FUNCTION_BLOCK FB_CommandInvoker
VAR_GENERIC CONSTANT
	CommandCapacity : UINT := 10;
END_VAR
EXTENDS FB_Base
VAR
	_Commands : ARRAY[0..CommandCapacity - 1] OF I_Command;
	_CommandCount : UINT;
	
	_InvokeIndex : UINT;
	_ProgressState : E_Progress;
	
	_PauseRequest : BOOL;
	_StepMode : BOOL;
END_VAR

METHOD AddCommand : BOOL
VAR_INPUT
	command : I_Command;
END_VAR
IF (NOT _CommandCount < CommandCapacity) THEN
	Tc2_System.ADSLOGSTR(0, 'Can not add any more commands!', '');
	RETURN;
END_IF

_Commands[_CommandCount] := command;
_CommandCount := _CommandCount + 1;

AddCommand := TRUE;
END_METHOD

METHOD ClearCommands
VAR
	i : UINT;
	p : POINTER TO BYTE;
END_VAR
FOR i := 0 TO _CommandCount - 1 DO
	__QUERYPOINTER(_Commands[i], p);
	__DELETE(p);
END_FOR

_CommandCount := 0;
END_METHOD

{attribute 'monitoring' := 'call'}
PROPERTY CommandCount : UINT
GET
CommandCount := _CommandCount;
END_GET
END_PROPERTY

{attribute 'monitoring' := 'call'}
PROPERTY Commands : REFERENCE TO ARRAY[0..CommandCapacity - 1] OF I_Command
GET
Commands REF= _Commands;
END_GET
END_PROPERTY

METHOD Cyclic
VAR_INPUT
END_VAR
IF (_ProgressState = E_Progress.Running) THEN
	Invoke();
END_IF
END_METHOD

//FB_Exit must be implemented explicitly. If there is an implementation, then the
//method is called before the controller removes the code of the function block instance
//(implicit call). The return value is not evaluated.
METHOD FB_Exit: BOOL
VAR_INPUT
    bInCopyCode: BOOL;  // TRUE: the exit method is called in order to leave the instance which will be copied afterwards (online change).  
END_VAR
ClearCommands();
END_METHOD

METHOD PRIVATE Invoke
VAR
	commandProgress : E_Progress;
	progress : T_MaxString;
	test : STRING := 'test';
END_VAR
IF (_CommandCount = 0) THEN
	_ProgressState := E_Progress.Completed;
	
	Tc2_System.ADSLOGSTR(0, 'Invoker finished. No commands were executed.', '');	
END_IF

IF (_InvokeIndex < _CommandCount) THEN
	
	commandProgress := _Commands[_InvokeIndex].Execute();
	IF (commandProgress = E_Progress.Completed) THEN
		
		IF (_PauseRequest OR _StepMode) THEN
			_ProgressState := E_Progress.Paused;
			_PauseRequest := FALSE;
		END_IF
		
		IF (_InvokeIndex = _CommandCount - 1) THEN
			_ProgressState := E_Progress.Completed;
			
			Tc2_System.ADSLOGSTR(0, 'Invoker finished', '');
		END_IF

		_InvokeIndex := _InvokeIndex + 1;
		
		progress := 'Invoker progress  ';
		progress := CONCAT(progress, TO_STRING(_InvokeIndex));
		progress := CONCAT(progress, '/');
		progress := CONCAT(progress, TO_STRING(_CommandCount));
		progress := CONCAT(progress, '  ');
		progress := CONCAT(progress, LREAL_TO_FMTSTR(ProgressPercent, 1, TRUE));
		progress := CONCAT(progress, ' %s');
		Tc2_System.ADSLOGSTR(0, progress, '%');
// 		Tc2_System.ADSLOGSTR(0, 'ahoj', '');
// 		Tc2_System.ADSLOGSTR(0, progress, '');
	END_IF
END_IF
END_METHOD

{attribute 'monitoring' := 'call'}
PROPERTY InvokeIndex : UINT
GET
InvokeIndex := _InvokeIndex;
END_GET
END_PROPERTY

METHOD Pause
VAR_INPUT
END_VAR
_PauseRequest := TRUE;
END_METHOD

{attribute 'monitoring' := 'call'}
PROPERTY PauseRequest : BOOL
GET
PauseRequest := _PauseRequest;
END_GET
END_PROPERTY

{attribute 'monitoring' := 'call'}
PROPERTY ProgressPercent : REAL
GET
IF (_CommandCount > 0) THEN
	ProgressPercent := 100.0 * _InvokeIndex / _CommandCount;
ELSE
	ProgressPercent := 0;
END_IF
END_GET
END_PROPERTY

{attribute 'monitoring' := 'call'}
PROPERTY ProgressState : E_Progress
GET
ProgressState := _ProgressState;
END_GET
END_PROPERTY

METHOD Reset
VAR_INPUT
END_VAR
_InvokeIndex := 0;
_ProgressState := E_Progress.Idle;

_PauseRequest := FALSE;
END_METHOD

METHOD Start
VAR_INPUT
END_VAR
CASE _ProgressState OF
	
	E_Progress.Idle,
	E_Progress.Paused,
	E_Progress.Completed:
		
		IF (NOT(_ProgressState = E_Progress.Paused
				OR (_ProgressState = E_Progress.Running AND (_PauseRequest OR _StepMode)))) THEN
			
			_InvokeIndex := 0;
		END_IF
		
		_ProgressState := E_Progress.Running;
		_PauseRequest := FALSE;

		Tc2_System.ADSLOGSTR(0, 'Invoker started', '');
END_CASE
END_METHOD

{attribute 'monitoring' := 'call'}
PROPERTY StepMode : BOOL
GET
StepMode := _StepMode;
END_GET
SET
_StepMode := StepMode;
END_SET
END_PROPERTY

END_FUNCTION_BLOCK

(* stored: Version 1.1.0.1
   POU FB_CommandInvoker: Id {f6ea97c1-b361-4680-9d27-e17b57602f50}, SpecialFunc None
   Method AddCommand: Id {558a4463-945b-4535-b113-75c835b88ed2}
   Method ClearCommands: Id {9a94bee6-4b43-4ebc-88ec-031ddc3491a8}
   Property CommandCount: Id {d512b632-5a54-480f-9bce-4617787f69fe}
   Get Get: Id {284783af-223d-4d79-a2b0-d4621b790078}
   Property Commands: Id {2ac8551e-9166-43fb-bc1a-2591e3449bd0}
   Get Get: Id {7c052ed9-b4b8-4aba-bf27-d5e3facd9369}
   Method Cyclic: Id {3cedf336-2bc5-4fe9-9158-43b939c09fe9}
   Method FB_Exit: Id {8216066f-20db-4c2b-b4a5-5d35467c67e9}
   Method Invoke: Id {1fb6d0da-5c0e-4695-bca1-1392766a0f71}
   Property InvokeIndex: Id {ed028e02-57f8-4247-bc34-7a9644dd0787}
   Get Get: Id {a1d3390e-bce7-44b8-86fd-ea6ad8635a83}
   Method Pause: Id {60346052-1c5c-4869-852f-cee975ff6538}
   Property PauseRequest: Id {e2ed5e62-1210-44f6-b001-af23576cae5d}
   Get Get: Id {be2f6951-47a5-42fc-80f5-fb5ed713bbd3}
   Property ProgressPercent: Id {a1b66641-0dc1-42f7-9b6f-b32b2a7e9dbc}
   Get Get: Id {05699fa0-c139-4e87-a24b-14be290e1b8e}
   Property ProgressState: Id {9ad5fd53-3f56-4334-a0c6-c35562f308f3}
   Get Get: Id {40a75a82-8678-4c39-9502-b446977d447b}
   Method Reset: Id {e85a53c0-fd47-4631-ae26-653508aa1e43}
   Method Start: Id {07470539-7ede-4172-96a9-a7980587ec0b}
   Property StepMode: Id {8cddf28e-f041-4432-90df-0de57b23caaf}
   Get Get: Id {329dfed4-6231-4420-8c66-6b4c744a4c62}
   Set Set: Id {cf9bb55f-41ba-4494-a585-3446254d6539} *)
